PROGRAM Rep_Bs
VAR
	FB_B1572_Rep_Bs	:FB_Rep_Ethercat_MURR;
	//FC inclure en port X6 EV Serr/Desserr guide coupe fer
	
END_VAR

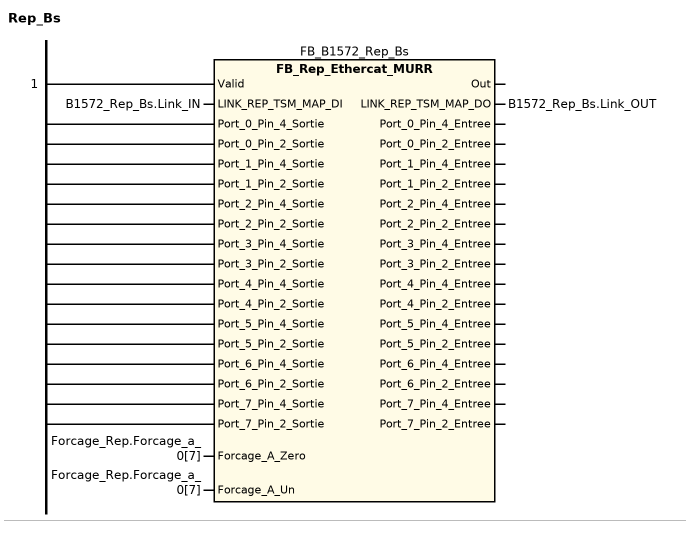
// NETWORK 1
FB_B1572_Rep_Bs(
    Valid := TRUE,
    LINK_REP_TSM_MAP_DI := B1572_Rep_Bs.Link_IN,
    Port_0_Pin_4_Sortie := TRUE,
    Port_0_Pin_2_Sortie := TRUE,
    Port_1_Pin_4_Sortie := TRUE,
    Port_1_Pin_2_Sortie := TRUE,
    Port_2_Pin_4_Sortie := TRUE,
    Port_2_Pin_2_Sortie := TRUE,
    Port_3_Pin_4_Sortie := TRUE,
    Port_3_Pin_2_Sortie := TRUE,
    Port_4_Pin_4_Sortie := TRUE,
    Port_4_Pin_2_Sortie := TRUE,
    Port_5_Pin_4_Sortie := TRUE,
    Port_5_Pin_2_Sortie := TRUE,
    Port_6_Pin_4_Sortie := TRUE,
    Port_6_Pin_2_Sortie := TRUE,
    Port_7_Pin_4_Sortie := TRUE,
    Port_7_Pin_2_Sortie := TRUE,
    Forcage_A_Zero := Forcage_Rep.Forcage_a_0[7],
    Forcage_A_Un := Forcage_Rep.Forcage_a_0[7],
    LINK_REP_TSM_MAP_DO => B1572_Rep_Bs.Link_OUT); // FB_Rep_Ethercat_MURR

END_PROGRAM

(* stored: Version 1.1.0.1
   POU Rep_Bs: Id {3dde847b-7644-4940-8bb9-5d4dc303a434}, SpecialFunc None *)
